(* Logix 5000 project; controller PLCbox vendor 1 type 14 code 149 rev 30.11; software revision 30.01 *)

TASK MainTask (continuous, watchdog 500 ms) : MainProgram, TestProgram, ExternalHardware
TASK Projects (periodic, rate 10 ms, priority 10, watchdog 500 ms) : StreetLightSystem
TASK ST_Routines (periodic, rate 10 ms, priority 10, watchdog 500 ms) : ST_Practice
TASK Task100msec (periodic, rate 100 ms, priority 2, watchdog 500 ms) : MainProgram2
TASK Tutorials (periodic, rate 10 ms, priority 10, watchdog 500 ms) : Mathematical, InterviewPractice, CognexJobChange, Challenges_Projects, TankFillingChallenge, FTViewTutorial, Advanced

MODULES
   Local : vendor 1 type 14 code 149 (Compact 0, rev 30.11)
      Discrete_IO : Embedded (Compact 1, rev 3.1, Output RPI 20 ms)
      CLX_PLC : 1756-EN2T (Ethernet 192.168.1.30, rev 5.28)
         CLX_MainPLC : vendor 1 type 14 code 54 (ICP 0, rev 20.4, $1bb2e967$ RPI 20 ms)
      VladCognex : vendor 678 type 100 code 265 (Ethernet 192.168.1.15, rev 4.10, Output RPI 20 ms)
      PointIO_Rack1 : 1734-AENT (Ethernet 192.168.1.9, rev 5.12, Output RPI 20 ms)
         Rem_IN_1 : 1734-IB8 (PointIO 1, rev 3.1)
         Rem_IN_2 : 1734-IB8 (PointIO 2, rev 3.1)
         Rem_OUT_3 : 1734-OB8E (PointIO 3, rev 3.1)
END_MODULES

TYPE String20 :
STRUCT
   LEN : DINT;
   DATA : SINT[20];
END_STRUCT
END_TYPE

TYPE UDT_Output :
STRUCT
   Energize : BOOL;
   Auto : BOOL;
   ManualAvl : BOOL;
   Force : BOOL;
   ForceAvl : BOOL;
   Delay_ON : TIMER;
   Name : String20;
   SetAuto : BOOL;
   SetManual : BOOL;
   ForceON : BOOL;
   ForceOFF : BOOL;
END_STRUCT
END_TYPE

TYPE UDT_PID :
STRUCT
   P : REAL;
   I : REAL;
   D : REAL;
   CV : REAL;
   SP : REAL;
   PV : REAL;
   Auto : BOOL;
   Name : STRING;
END_STRUCT
END_TYPE

TYPE UDT_ProdCons :
STRUCT
   Status : CONNECTION_STATUS;
   Data : DINT[50];
END_STRUCT
END_TYPE

TYPE UDT_Time :
STRUCT
   Year : DINT;
   Month : DINT;
   Day : DINT;
   Hour : DINT;
   Minute : DINT;
   Second : DINT;
   Microsecond : DINT;
END_STRUCT
END_TYPE

ADD_ON_INSTRUCTION AOI_BasicCalculation   (* revision 1.0, vendor SolisPLC *)
VAR_INPUT
   Operand_1 : REAL; {required}
   Operand_2 : REAL; {required}
   Operand_3 : REAL; {required}
   Operand_4 : REAL; {required}
END_VAR
VAR_OUTPUT
   Multiplication : REAL; {access Read Only, required}
   Addition : REAL; {access Read Only, required}
END_VAR
VAR
   Mul1 : REAL; {access None}
   Mul2 : REAL; {access None}
   Add1 : REAL; {access None}
   Add2 : REAL; {access None}
END_VAR

ROUTINE Logic   (* ladder *)
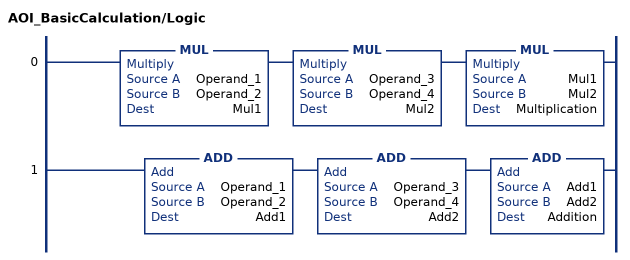
   0: MUL(Operand_1,Operand_2,Mul1)MUL(Operand_3,Operand_4,Mul2)MUL(Mul1,Mul2,Multiplication);
   1: ADD(Operand_1,Operand_2,Add1)ADD(Operand_3,Operand_4,Add2)ADD(Add1,Add2,Addition);
END_ROUTINE
END_ADD_ON_INSTRUCTION

VAR_GLOBAL   (* controller tags *)
   BNOT_1501 : FBD_BOOLEAN_NOT := (In := 1);
   CLX_Cons : UDT_ProdCons := (Status.ConnectionFaulted := 1);
   CMPLX_Prod : UDT_ProdCons := (Status.RunMode := 1, Data[0] := 56789, Data[5] := 674); {produced}
   HMI_Int_BOOL : BOOL[64] := ([2] := 1, [3] := 1);
        [0]   // Light 1 Status - Green
        [1]   // Light 1 Status - Yellow
        [2]   // Light 1 Status - Red
        [3]   // Light 2 Status - Green
        [4]   // Light 2 Status - Yellow
        [5]   // Light 2 Status - Red
   HMI_Interface_BOOL : BOOL[64];
        [0]   // Light 1 - Green Status ON
        [1]   // Light 1 - Yellow Status ON
        [2]   // Light 1 - Red Status ON
        [3]   // Light 2 - Green Status ON
        [4]   // Light 2 - Yellow Status ON
        [5]   // Light 2 - Red Status ON
   HMI_No_Access : BOOL;
   IN_Loc1 : BOOL[32];
        [0]   // Local Input 1 - Green Pushbutton ON
        [1]   // Local Input 2 - Yellow Pushbutton ON
        [2]   // Local Input 3 - Motor 1 Running
   IN_Loc1_DB_OFF : BOOL[32];
   IN_Loc1_DB_ON : BOOL[32];
   IN_Loc1_Index : DINT := 16;
   IN_Loc1_T_OFF : TIMER[16] := ([0].PRE := 500, [0].ACC := 500);
   IN_Loc1_T_ON : TIMER[16] := ([0].PRE := 500);
   JobData : SINT[32] := ([0] := 16, [2] := 70, [3] := 105, [4] := 114, [5] := 115, [6] := 116, [7] := 74, [8] := 111, [9] := 98, [10] := 84, [11] := 101, [12] := 115, [13] := 116, [14] := 46, [15] := 106, [16] := 111, [17] := 98);
   Light1_Complete_ONS : BOOL := 1;
   Light1_Green : BOOL;
   Light1_Green_T : TIMER := (PRE := 10000, ACC := 10000, EN := 1, DN := 1);
   Light1_Red : BOOL := 1;
   Light1_Reset : BOOL;
   Light1_Yellow : BOOL;
   Light1_Yellow_T : TIMER := (PRE := 3000, ACC := 3000, EN := 1, DN := 1);
   Light2_Complete_ONS : BOOL;
   Light2_Green : BOOL := 1;
   Light2_Green_T : TIMER := (PRE := 10000, ACC := 1060, EN := 1, TT := 1);
   Light2_Red : BOOL;
   Light2_Reset : BOOL;
   Light2_Yellow : BOOL;
   Light2_Yellow_T : TIMER := (PRE := 3000);
   NewProductID : DINT := 1017;
   OUT_Loc1 : BOOL[32] := ([0] := 1);
   PID_Analog_In : REAL[20];
   PLCTime : UDT_Time := (Year := 2019, Month := 5, Day := 7, Hour := 16, Minute := 4, Second := 58, Microsecond := 209573);
   SetJob : MESSAGE;
        MessageParameters(ServiceCode := 16#0010, LocalElement := JobData[0], ...)
   SsytemStopped : BOOL := 1;
   System_Timer : TIMER[100] := ([0].PRE := 10000, [0].ACC := 1170, [0].EN := 1, [0].TT := 1);
   tagToPi : DINT := 1010;
   TIC_1501 : PID_ENHANCED := (PVEUMax := 100.0, SPHLimit := 100.0, RatioProg := 1.0, RatioOper := 1.0, RatioHLimit := 1.0, RatioLLimit := 1.0, CVEUMax := 100.0, CVHLimit := 100.0, PVEDerivative := 1, RTSTime := 1);
END_VAR

PROGRAM Advanced   (* main routine _01_Main *)
VAR
   Add : REAL;
   AOI_Basic1 : AOI_BasicCalculation;
   Mult : REAL;
   Op1 : REAL;
   Op2 : REAL;
   Op3 : REAL;
   Op4 : REAL;
   PLCCond : BOOL[32];
   PLCCondOut : BOOL[32] := ([1] := 1);
   SeqArr : DINT[10] := ([0] := 1, [1] := 2, [2] := 4, [3] := 8);
   SeqArr2 : DINT[10] := ([0] := 1, [1] := 2, [2] := 4, [3] := 8, [4] := 16);
   SeqControl : CONTROL := (LEN := 3, POS := 1);
   SeqMask : DINT := 15;
   SeqOut : DINT := 2;
   SeqSource : DINT;
END_VAR

ROUTINE _01_Main   (* ladder *)
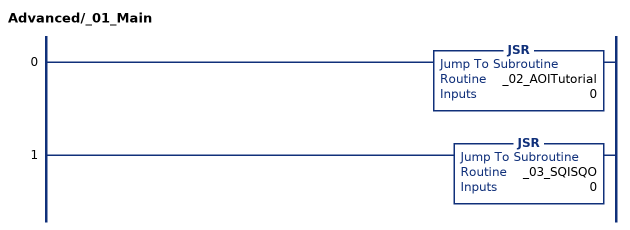
   0: JSR(_02_AOITutorial,0);
   1: JSR(_03_SQISQO,0);
END_ROUTINE

ROUTINE _02_AOITutorial   (* ladder *)
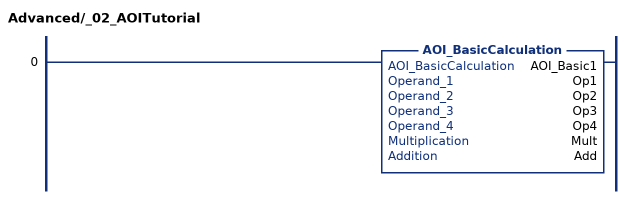
   0: AOI_BasicCalculation(AOI_Basic1,Op1,Op2,Op3,Op4,Mult,Add);
END_ROUTINE

ROUTINE _03_SQISQO   (* ladder *)
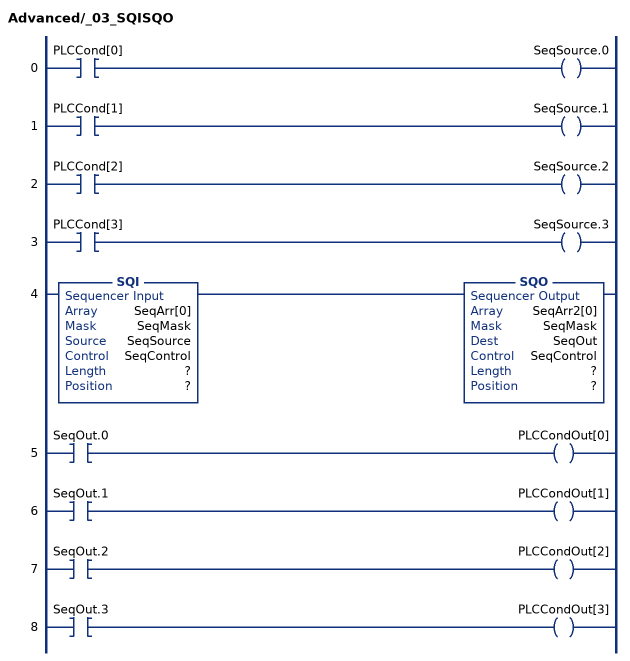
   0: XIC(PLCCond[0])OTE(SeqSource.0);
   1: XIC(PLCCond[1])OTE(SeqSource.1);
   2: XIC(PLCCond[2])OTE(SeqSource.2);
   3: XIC(PLCCond[3])OTE(SeqSource.3);
   4: SQI(SeqArr[0],SeqMask,SeqSource,SeqControl,?,?)SQO(SeqArr2[0],SeqMask,SeqOut,SeqControl,?,?);
   5: XIC(SeqOut.0)OTE(PLCCondOut[0]);
   6: XIC(SeqOut.1)OTE(PLCCondOut[1]);
   7: XIC(SeqOut.2)OTE(PLCCondOut[2]);
   8: XIC(SeqOut.3)OTE(PLCCondOut[3]);
END_ROUTINE
END_PROGRAM

PROGRAM Challenges_Projects   (* main routine _01_Main *)
VAR
   GREEN_LIGHT_ON : BOOL;
   RED_LIGHT_ON : BOOL;
   RESET_PRESSED : BOOL;
   START_PRESSED : BOOL;
   STOP_PRESSED : BOOL;
   YELLOW_LIGHT_ON : BOOL;
END_VAR

ROUTINE _01_Main   (* ladder *)
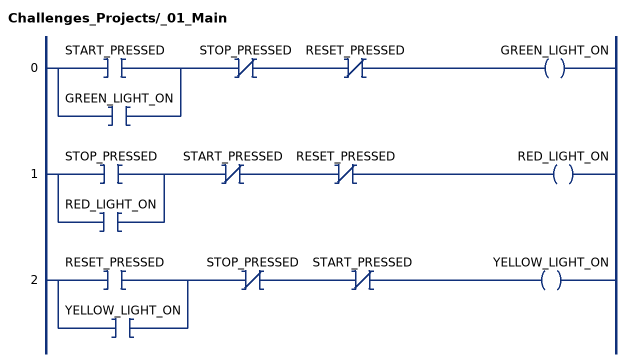
   0: [XIC(START_PRESSED) ,XIC(GREEN_LIGHT_ON) ]XIO(STOP_PRESSED)XIO(RESET_PRESSED)OTE(GREEN_LIGHT_ON);
   1: [XIC(STOP_PRESSED) ,XIC(RED_LIGHT_ON) ]XIO(START_PRESSED)XIO(RESET_PRESSED)OTE(RED_LIGHT_ON);
   2: [XIC(RESET_PRESSED) ,XIC(YELLOW_LIGHT_ON) ]XIO(STOP_PRESSED)XIO(START_PRESSED)OTE(YELLOW_LIGHT_ON);
END_ROUTINE
END_PROGRAM

PROGRAM CognexJobChange   (* main routine Main *)
VAR
   JobIndex : DINT := 1;
   JobName : STRING[10] := ([0] := 'VladsJob.job', [1] := 'FirstJobTest.job', [2] := 'BarcodeRead.job');
   JobSet : BOOL[32];
   JobTrigger : BOOL;
   TriggerONS : BOOL;
   VladsCounter : COUNTER := (ACC := 11, DN := 1);
END_VAR

ROUTINE Main   (* ladder *)
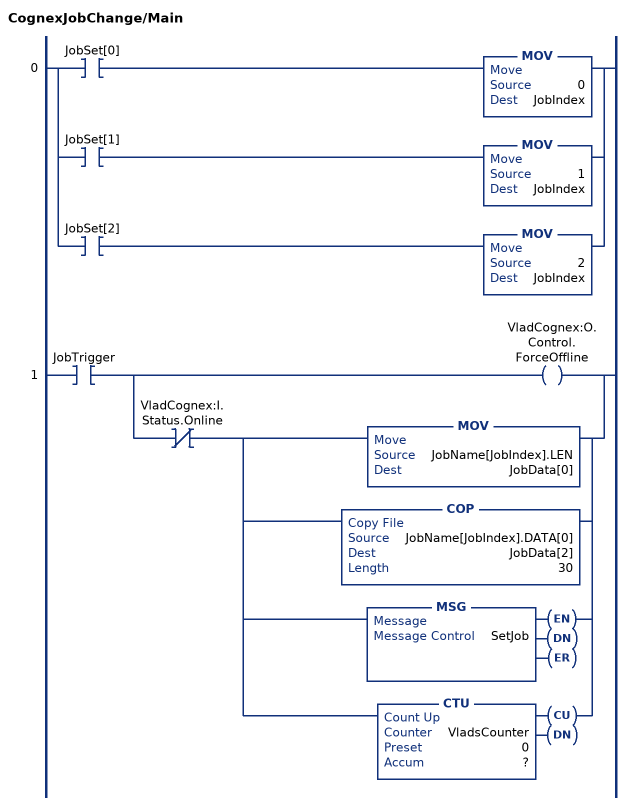
   0: [XIC(JobSet[0]) MOV(0,JobIndex) ,XIC(JobSet[1]) MOV(1,JobIndex) ,XIC(JobSet[2]) MOV(2,JobIndex) ];
   1: XIC(JobTrigger)[OTE(VladCognex:O.Control.ForceOffline) ,XIO(VladCognex:I.Status.Online) [MOV(JobName[JobIndex].LEN,JobData[0]) ,COP(JobName[JobIndex].DATA[0],JobData[2],30) ,MSG(SetJob) ,CTU(VladsCounter,?,?) ] ];
END_ROUTINE
END_PROGRAM

PROGRAM ExternalHardware   (* main routine _01_Main *)
VAR
   HMI_O_Screeen_Title : String20[100] := ([0] := 'Slot 0 - Local Out.', [1] := 'Main Screen', [2] := 'System Settings', [3] := 'In Q - Motor Starter', [4] := 'Alarm Display');
END_VAR

ROUTINE _01_Main   (* ladder *)
END_ROUTINE
END_PROGRAM

PROGRAM FTViewTutorial   (* main routine _01_Main *)
VAR
   AlarmReset : BOOL;
   HMI_Rotation : TIMER := (PRE := 5000, ACC := 2560, EN := 1, TT := 1);
   HMI_Rotation_Enable : BOOL := 1;
   Motor1HL : BOOL;
   Motor1LL : BOOL;
   Motor1Speed : REAL := 60.0;
   Motor1SpeedActual : REAL := 60.0;
   Motor1SpeedSetpoint : REAL := 60.0;
   Motor1Var : REAL := 5.0;
END_VAR

ROUTINE _01_Main   (* ladder *)
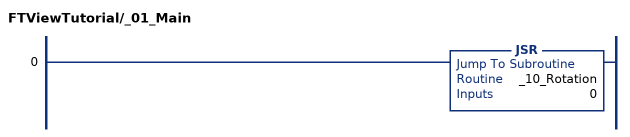
   0: JSR(_10_Rotation,0);
END_ROUTINE

ROUTINE _10_Rotation   (* ladder *)
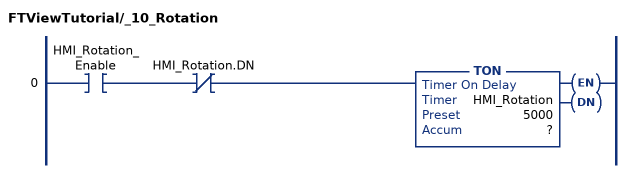
   0: XIC(HMI_Rotation_Enable)XIO(HMI_Rotation.DN)TON(HMI_Rotation,?,?);
END_ROUTINE
END_PROGRAM

PROGRAM InterviewPractice   (* main routine _01_Main *)
VAR
   INT_Motor : BOOL[32];
        [0]   // START
        [10]   // MOTOR STARTER
        [1]   // STOP
        [2]   // MOTOR OVERLOAD / FAULT
END_VAR

ROUTINE _01_Main   (* ladder *)
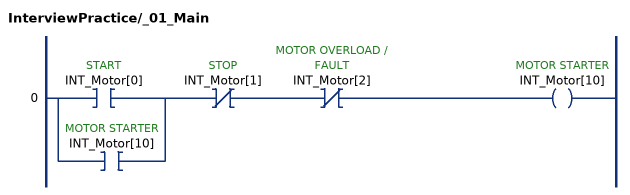
   0: [XIC(INT_Motor[0]) ,XIC(INT_Motor[10]) ]XIO(INT_Motor[1])XIO(INT_Motor[2])OTE(INT_Motor[10]);
END_ROUTINE
END_PROGRAM

PROGRAM MainProgram   (* main routine _01_Main *)
VAR
   ClearString : String20;
   FinalCode : String20 := '$00$00$00$00$00$00$00$00$00$00$00$00$C4$016$F1$00$00$00$00';
   LocalDebounceTimer : TIMER;
   LocInDebounced1 : BOOL;
   MFinalCode : String20 := 'VW$00$00$00$00$00$00$1C$00$00$80$C4$016$F1$00$00$00$00';
   MyBarcode : STRING := '$00$00$00$00$00$00$00$00$00$00$00$00$C4$016$F1$00$00$00$00$CE$8F$0A$00X$00$00$0063013337$0A$00$00$80$1C$00$00$80$C4$016$F1$00$00$00$00$CE$8F$0A$00X$00$00$0063013337$0A$00$00$80$1C$00$00$80$C4$016$F1$00$00$00$00';
   OUT_Loc1_AUTO : BOOL[32] := ([0] := 1, [1] := 1, [2] := 1, [3] := 1, [4] := 1, [5] := 1, [6] := 1, [7] := 1, [8] := 1, [9] := 1, [10] := 1, [11] := 1, [12] := 1, [13] := 1, [14] := 1, [15] := 1, [16] := 1, [17] := 1, [18] := 1, [19] := 1, [20] := 1, [21] := 1, [22] := 1, [23] := 1, [24] := 1, [25] := 1, [26] := 1, [27] := 1, [28] := 1, [29] := 1, [30] := 1, [31] := 1);
   OUT_Loc1_F : BOOL[32] := ([0] := 1);
   OUT_Loc1_Final : BOOL;
   OUT_Loc1_FORCE : BOOL[32];
   OUT_Loc1_Index : DINT := 16;
   OUT_S1 : UDT_Output[16] := ([0].Auto := 1, [0].ManualAvl := 1, [0].Name := 'Test Tag', [1].Auto := 1, [1].ManualAvl := 1, [2].Auto := 1, [2].ManualAvl := 1, [3].ManualAvl := 1, [3].ForceAvl := 1, [4].Auto := 1, [4].ManualAvl := 1, [5].ManualAvl := 1, [5].ForceAvl := 1, [6].ManualAvl := 1, [6].ForceAvl := 1, [7].ManualAvl := 1, [7].ForceAvl := 1, [8].ManualAvl := 1, [8].ForceAvl := 1, [9].Auto := 1, [9].ManualAvl := 1, [10].Auto := 1, [10].ManualAvl := 1, [11].ManualAvl := 1, [11].ForceAvl := 1, [12].ManualAvl := 1, [12].ForceAvl := 1, [13].ManualAvl := 1, [13].ForceAvl := 1, [14].ManualAvl := 1, [14].ForceAvl := 1, [15].ManualAvl := 1, [15].ForceAvl := 1);
   STR : STRING := '825242422';
   test : DINT := 825242422;
   test2 : DINT[2];
END_VAR

ROUTINE _01_Main   (* ladder *)
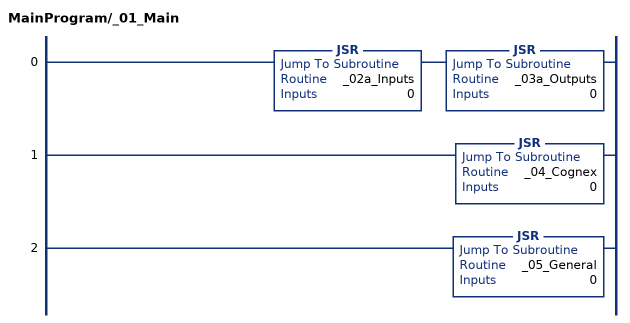
   0: JSR(_02a_Inputs,0)JSR(_03a_Outputs,0);
   1: JSR(_04_Cognex,0);
   2: JSR(_05_General,0);
END_ROUTINE

ROUTINE _02a_Inputs   (* ladder *)
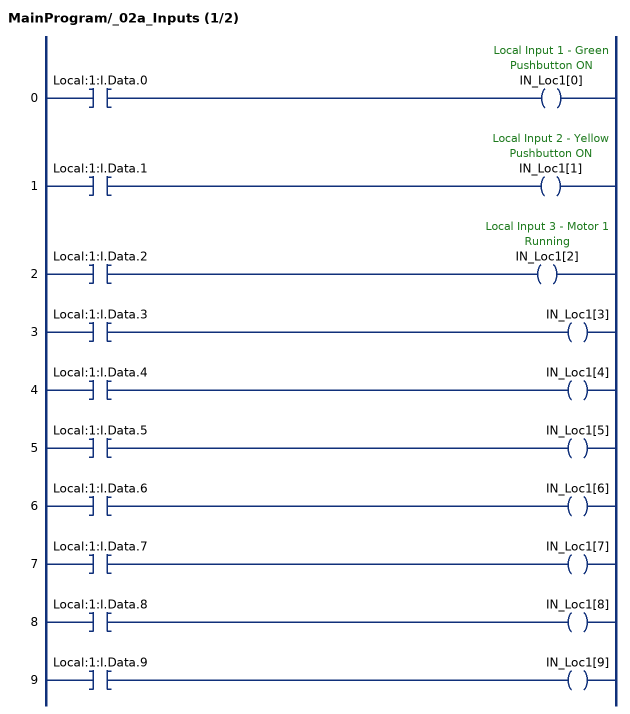
   0: XIC(Local:1:I.Data.0)OTE(IN_Loc1[0]);
   1: XIC(Local:1:I.Data.1)OTE(IN_Loc1[1]);
   2: XIC(Local:1:I.Data.2)OTE(IN_Loc1[2]);
   3: XIC(Local:1:I.Data.3)OTE(IN_Loc1[3]);
   4: XIC(Local:1:I.Data.4)OTE(IN_Loc1[4]);
   5: XIC(Local:1:I.Data.5)OTE(IN_Loc1[5]);
   6: XIC(Local:1:I.Data.6)OTE(IN_Loc1[6]);
   7: XIC(Local:1:I.Data.7)OTE(IN_Loc1[7]);
   8: XIC(Local:1:I.Data.8)OTE(IN_Loc1[8]);
   9: XIC(Local:1:I.Data.9)OTE(IN_Loc1[9]);
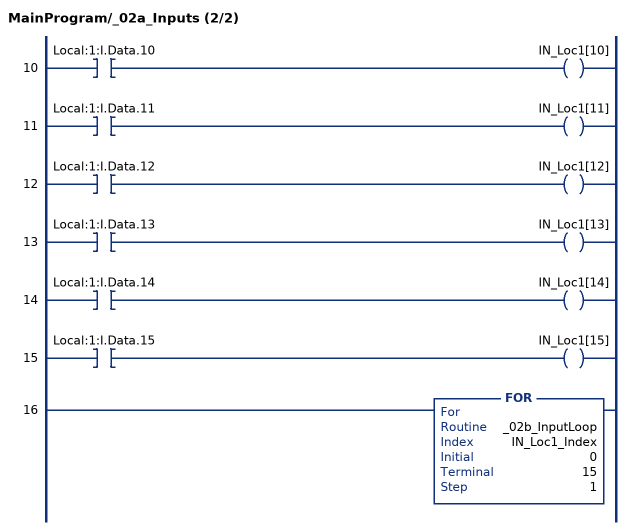
   10: XIC(Local:1:I.Data.10)OTE(IN_Loc1[10]);
   11: XIC(Local:1:I.Data.11)OTE(IN_Loc1[11]);
   12: XIC(Local:1:I.Data.12)OTE(IN_Loc1[12]);
   13: XIC(Local:1:I.Data.13)OTE(IN_Loc1[13]);
   14: XIC(Local:1:I.Data.14)OTE(IN_Loc1[14]);
   15: XIC(Local:1:I.Data.15)OTE(IN_Loc1[15]);
   16: FOR(_02b_InputLoop,IN_Loc1_Index,0,15,1);
END_ROUTINE

ROUTINE _02b_InputLoop   (* ladder *)
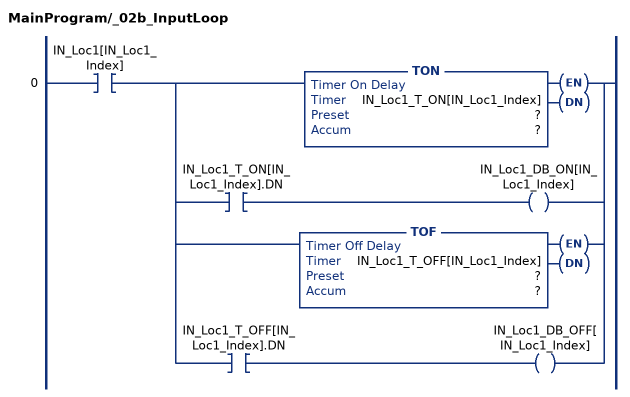
   0: XIC(IN_Loc1[IN_Loc1_Index])[TON(IN_Loc1_T_ON[IN_Loc1_Index],?,?) ,XIC(IN_Loc1_T_ON[IN_Loc1_Index].DN) OTE(IN_Loc1_DB_ON[IN_Loc1_Index]) ,TOF(IN_Loc1_T_OFF[IN_Loc1_Index],?,?) ,XIC(IN_Loc1_T_OFF[IN_Loc1_Index].DN) OTE(IN_Loc1_DB_OFF[IN_Loc1_Index]) ];
END_ROUTINE

ROUTINE _03a_Outputs   (* ladder *)
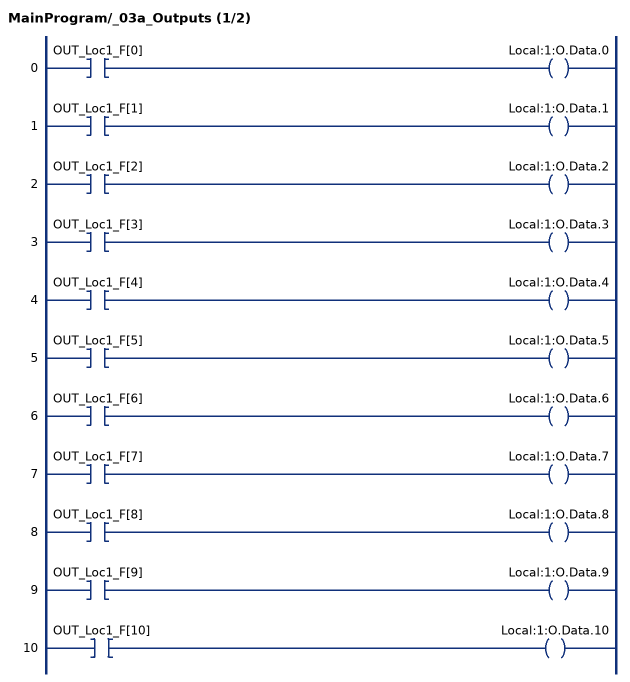
   0: XIC(OUT_Loc1_F[0])OTE(Local:1:O.Data.0);
   1: XIC(OUT_Loc1_F[1])OTE(Local:1:O.Data.1);
   2: XIC(OUT_Loc1_F[2])OTE(Local:1:O.Data.2);
   3: XIC(OUT_Loc1_F[3])OTE(Local:1:O.Data.3);
   4: XIC(OUT_Loc1_F[4])OTE(Local:1:O.Data.4);
   5: XIC(OUT_Loc1_F[5])OTE(Local:1:O.Data.5);
   6: XIC(OUT_Loc1_F[6])OTE(Local:1:O.Data.6);
   7: XIC(OUT_Loc1_F[7])OTE(Local:1:O.Data.7);
   8: XIC(OUT_Loc1_F[8])OTE(Local:1:O.Data.8);
   9: XIC(OUT_Loc1_F[9])OTE(Local:1:O.Data.9);
   10: XIC(OUT_Loc1_F[10])OTE(Local:1:O.Data.10);
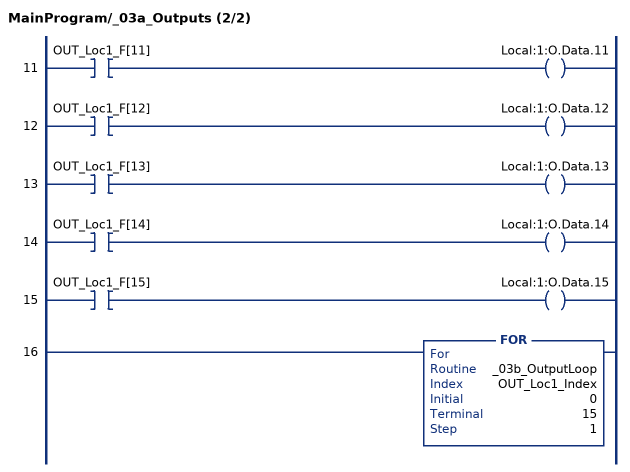
   11: XIC(OUT_Loc1_F[11])OTE(Local:1:O.Data.11);
   12: XIC(OUT_Loc1_F[12])OTE(Local:1:O.Data.12);
   13: XIC(OUT_Loc1_F[13])OTE(Local:1:O.Data.13);
   14: XIC(OUT_Loc1_F[14])OTE(Local:1:O.Data.14);
   15: XIC(OUT_Loc1_F[15])OTE(Local:1:O.Data.15);
   16: FOR(_03b_OutputLoop,OUT_Loc1_Index,0,15,1);
END_ROUTINE

ROUTINE _03b_OutputLoop   (* ladder *)
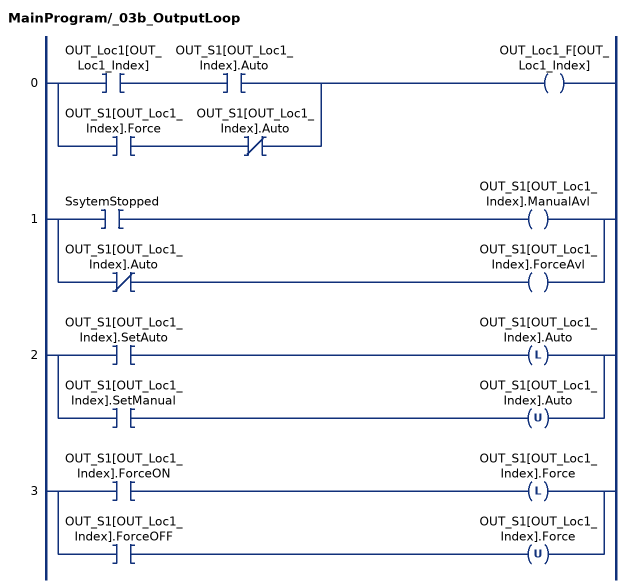
   0: [XIC(OUT_Loc1[OUT_Loc1_Index]) XIC(OUT_S1[OUT_Loc1_Index].Auto) ,XIC(OUT_S1[OUT_Loc1_Index].Force) XIO(OUT_S1[OUT_Loc1_Index].Auto) ]OTE(OUT_Loc1_F[OUT_Loc1_Index]);
   1: [XIC(SsytemStopped) OTE(OUT_S1[OUT_Loc1_Index].ManualAvl) ,XIO(OUT_S1[OUT_Loc1_Index].Auto) OTE(OUT_S1[OUT_Loc1_Index].ForceAvl) ];
   2: [XIC(OUT_S1[OUT_Loc1_Index].SetAuto) OTL(OUT_S1[OUT_Loc1_Index].Auto) ,XIC(OUT_S1[OUT_Loc1_Index].SetManual) OTU(OUT_S1[OUT_Loc1_Index].Auto) ];
   3: [XIC(OUT_S1[OUT_Loc1_Index].ForceON) OTL(OUT_S1[OUT_Loc1_Index].Force) ,XIC(OUT_S1[OUT_Loc1_Index].ForceOFF) OTU(OUT_S1[OUT_Loc1_Index].Force) ];
END_ROUTINE

ROUTINE _04_Cognex   (* ladder *)
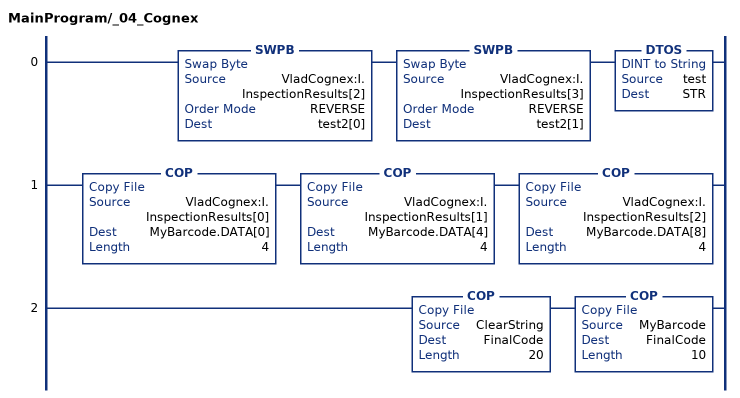
   0: SWPB(VladCognex:I.InspectionResults[2],REVERSE,test2[0])SWPB(VladCognex:I.InspectionResults[3],REVERSE,test2[1])DTOS(test,STR);
   1: COP(VladCognex:I.InspectionResults[0],MyBarcode.DATA[0],4)COP(VladCognex:I.InspectionResults[1],MyBarcode.DATA[4],4)COP(VladCognex:I.InspectionResults[2],MyBarcode.DATA[8],4);
   2: COP(ClearString,FinalCode,20)COP(MyBarcode,FinalCode,10);
END_ROUTINE

ROUTINE _05_General   (* ladder *)
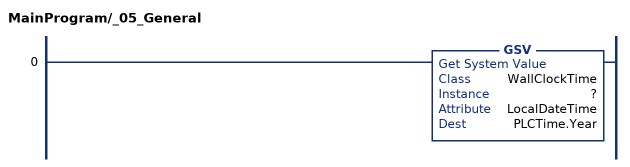
   0: GSV(WallClockTime,?,LocalDateTime,PLCTime.Year);
END_ROUTINE
END_PROGRAM
